FUNCTION_BLOCK SUB_3_LLP (* Dummy block for testing *)
  (* Standard: 61499-2 *)
  (* Version 0.0, 2002-12-17, JHC, Rockwell Automation, Copied from TEST_CAST *)
  (* Compiler header: package fb.rt.test; *)
  (* Compiler Java IBM JIkes 1.06 *)
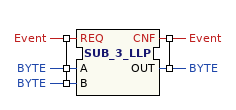
  EVENT_INPUT
    REQ WITH A, B; (* Normal Execution Request *)
  END_EVENT
  EVENT_OUTPUT
    CNF WITH OUT; (* Execution Confirmation *)
  END_EVENT
  VAR_INPUT
    A : BYTE;
    B : BYTE;
  END_VAR
  VAR_OUTPUT
    OUT : BYTE; (* A & B? *)
  END_VAR
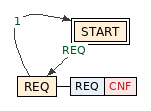
  EC_STATES
    START; (* Initial State *)
    REQ : REQ -> CNF; (* Normal execution *)
  END_STATES
  EC_TRANSITIONS
    START TO REQ := REQ;
    REQ TO START := 1;
  END_TRANSITIONS
  ALGORITHM REQ IN ST: (* Normally executed algorithm *)
OUT := A & B;
  END_ALGORITHM
END_FUNCTION_BLOCK
